{attribute 'linkalways'} 
{attribute 'no_explicit_call' := 'This FB is a CLASS and must be accessed using methods or properties'}
{attribute 'enable_dynamic_creation'}
FUNCTION_BLOCK FINAL AND_ULINT EXTENDS Node
VAR
	in1 : _ULINT(0);
	in2 : _ULINT(0);
	out : _ULINT(0);
END_VAR

METHOD PUBLIC Clone : I_Node
VAR
	pNode : POINTER TO AND_ULINT;
END_VAR
pNode := __NEW(AND_ULINT);
Clone := pNode^;
END_METHOD

METHOD FB_init : BOOL
VAR_INPUT
	bInitRetains : BOOL; // if TRUE, the retain variables are initialized (warm start / cold start)
	bInCopyCode : BOOL;  // if TRUE, the instance afterwards gets moved into the copy code (online change)
END_VAR
AddInput('in1',THIS^.in1);
AddInput('in2',THIS^.in2);
AddOutput('out', THIS^.out);
END_METHOD

METHOD PROTECTED OnExecute
VAR
END_VAR
out.Value := in1.Value AND in2.Value;
END_METHOD

END_FUNCTION_BLOCK

(* stored: Version 1.1.0.1, ProductVersion 3.1.4024.15
   POU AND_ULINT: Id {fee1575a-cfff-4984-82c4-87cd0b13c4ee}, SpecialFunc None
   Folder Constructor: Id {c5bd1f20-ffe1-41ec-b0f7-d014bff2dbb2}
   Method Clone: Id {56d2df29-85f7-4889-a8eb-af97934a60cd}
   Method FB_init: Id {e391bc85-9b16-41ff-945f-3ed5ea3055e9}
   Method OnExecute: Id {692d3191-108b-479b-81de-736888be539f} *)
